{attribute 'qualified_only'}
VAR_GLOBAL
	CartUp 			AT %Q*: BOOL := FALSE;		(* Lift kører op *)
	CartDown 		AT %Q*: BOOL := FALSE;		(* Lift kører ned *)
	CartForward 	AT %Q*: BOOL := FALSE;		(* Vogn kører fremad *)
	CartBackward 	AT %Q*: BOOL := FALSE;		(* Vogn kører bagud*)
	WheelsChange 	AT %Q*: BOOL := FALSE;		(* Hjul til sidelæns kørsel kører op/ned*)
END_VAR

(* stored: Version 1.1.0.1, ProductVersion 3.1.4024.4
   GVL CartControls: Id {b1b28d33-57c8-4051-a57c-80b215697c76} *)
